//structure includes unit information
TYPE ST_UnitInfo :
STRUCT
	Name		: STRING;
	ActState	: E_PMLState;
	ActMode		: DINT;
END_STRUCT
END_TYPE

(* stored: Version 1.1.0.1, ProductVersion 3.1.4018.5
   DUT ST_UnitInfo: Id {451caefe-2fbe-4f4f-b455-7197b6e77a1a} *)
